{attribute 'pack_mode' := '1'}
TYPE TDynAxisParam :
STRUCT
	Acc		: LREAL;
	Dec		: LREAL;
	Jerk		: LREAL;
END_STRUCT
END_TYPE

(* stored: Version 1.1.0.1, ProductVersion 3.1.4022.12
   DUT TDynAxisParam: Id {4cfd11a6-f9bc-4d95-848d-399c097cabbf} *)
